FUNCTION_BLOCK Button
  (* Standard: 61499-2 *)
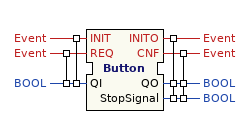
  EVENT_INPUT
    INIT WITH QI;
    REQ WITH QI;
  END_EVENT
  EVENT_OUTPUT
    INITO WITH QO, StopSignal;
    CNF WITH QO, StopSignal;
  END_EVENT
  VAR_INPUT
    QI : BOOL;
  END_VAR
  VAR_OUTPUT
    QO : BOOL;
    StopSignal : BOOL;
  END_VAR
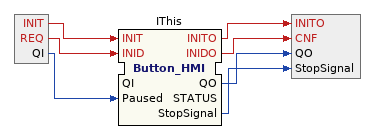
  FBS
    IThis : Button_HMI;
  END_FBS
  EVENT_CONNECTIONS
    INIT TO IThis.INIT;
    IThis.INITO TO INITO;
    IThis.INIDO TO CNF;
    REQ TO IThis.INID;
  END_CONNECTIONS
  DATA_CONNECTIONS
    IThis.StopSignal TO StopSignal;
    IThis.QO TO QO;
    QI TO IThis.Paused;
  END_CONNECTIONS
END_FUNCTION_BLOCK
